(* Schneider Machine Expert - Basic project M221_Program, file version 3.0.0.0 *)
(* ProjectInformations: Name=M221_Program *)

HARDWARE
  Cpu 0: TM221CE24T
  EthernetConfiguration: NetworkName=M221, IpAllocationMode=ByDhcp, IpAddress=192.168.1.10, SubnetMask=255.255.255.0
  SerialLineConfiguration: Baud=Baud19200, Parity=ParityEven, DataBits=DataBits8, StopBits=StopBits1, PhysicalMedium=PhysicalMediumRs485, TransmissionMode=TransmissionModeModbusRtu, SlaveId=1, Addressing=SlaveAddressing
  MastTask: UsePeriodScanMode=false, PeriodScan=100
  FastTask: Period=255
  CpuBehavior: StartingMode=StartAsPreviousState, AutoSaveRamOnEeprom=true, WatchdogPeriod=250

SYMBOLS  (address, symbol, comment, settings)
  %M0       TANK_FULL  "Tank is full"
  %M1       TANK_EMPTY  "Tank is empty"
  %Q0.0     INLET_VALVE
  %Q0.1     OUTLET_VALVE

POU Main Program
  (* SectionNumber=1 *)

// Rung 0: Tank Full Check
// Set TANK_FULL flag when level >= 3000mm
  LD [%IW1.0>=16000]
  ST %M0                  (* TANK_FULL *)
  // as ST:
  //   TANK_FULL := %IW1.0>=16000;
  (* the ladder stored for this rung does not match its IL; not drawn *)

// Rung 1: Tank Empty Check
// Set TANK_EMPTY flag when level <= 320mm
  LD [%IW1.0<=3200]
  ST %M1                  (* TANK_EMPTY *)
  // as ST:
  //   TANK_EMPTY := %IW1.0<=3200;
  (* the ladder stored for this rung does not match its IL; not drawn *)

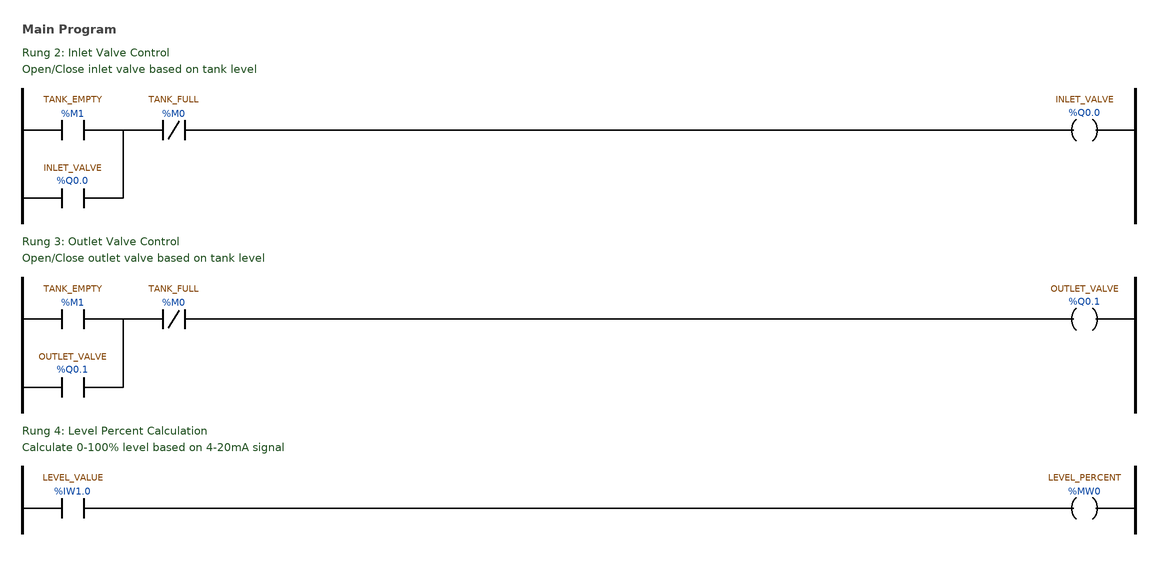

// Rung 2: Inlet Valve Control
// Open/Close inlet valve based on tank level
  LD %M1                  (* TANK_EMPTY *)
  OR %Q0.0                (* INLET_VALVE *)
  ANDN %M0                (* TANK_FULL *)
  ST %Q0.0                (* INLET_VALVE *)
  // as ST:
  //   INLET_VALVE := (TANK_EMPTY OR INLET_VALVE) AND NOT TANK_FULL;

// Rung 3: Outlet Valve Control
// Open/Close outlet valve based on tank level
  LD %M1                  (* TANK_EMPTY *)
  OR %Q0.1                (* OUTLET_VALVE *)
  ANDN %M0                (* TANK_FULL *)
  ST %Q0.1                (* OUTLET_VALVE *)
  // as ST:
  //   OUTLET_VALVE := (TANK_EMPTY OR OUTLET_VALVE) AND NOT TANK_FULL;

// Rung 4: Level Percent Calculation
// Calculate 0-100% level based on 4-20mA signal
  LD %IW1.0
  ST %MW0
  // as ST:
  //   %MW0 := %IW1.0;
